// Mitsubishi GX Works2 project: Rev 1   PLC: FX3G

PROGRAM MAIN
VAR
  b0 : BOOL;  (* Start Buttom *)
  b1 : BOOL;  (* Stop Button *)
  b2 : BOOL;  (* Refference Output *)
  sm400 : BOOL;
END_VAR
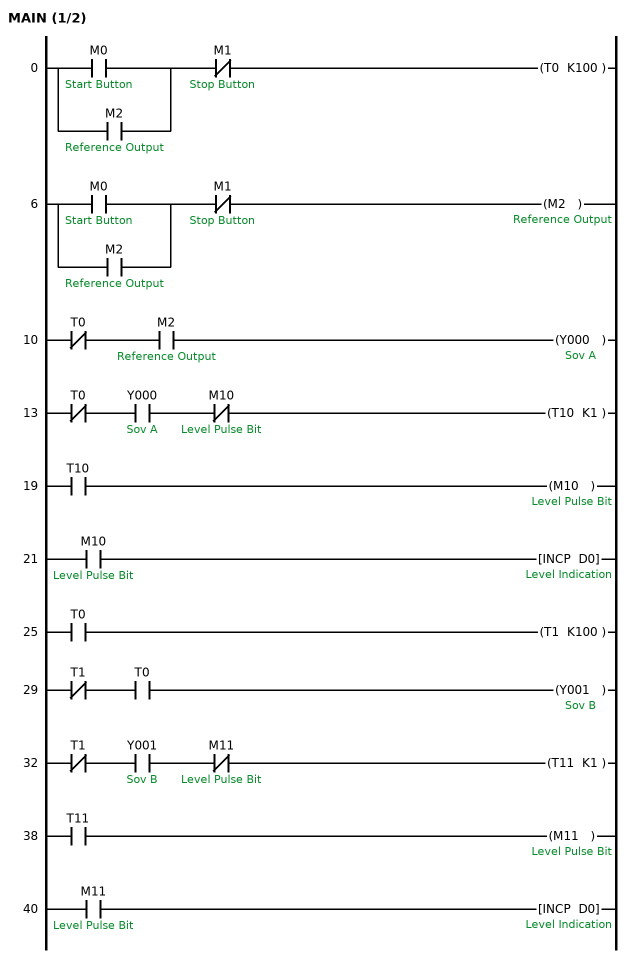
0     LD      M0  ; Start Button
      OR      M2  ; Reference Output
      ANI     M1  ; Stop Button
      OUT     T0 K100
6     LD      M0  ; Start Button
      OR      M2  ; Reference Output
      ANI     M1  ; Stop Button
      OUT     M2  ; Reference Output
10    LDI     T0
      AND     M2  ; Reference Output
      OUT     Y000  ; Sov A
13    LDI     T0
      AND     Y000  ; Sov A
      ANI     M10  ; Level Pulse Bit
      OUT     T10 K1
19    LD      T10
      OUT     M10  ; Level Pulse Bit
21    LD      M10  ; Level Pulse Bit
      INCP    D0  ; Level Indication
25    LD      T0
      OUT     T1 K100
29    LDI     T1
      AND     T0
      OUT     Y001  ; Sov B
32    LDI     T1
      AND     Y001  ; Sov B
      ANI     M11  ; Level Pulse Bit
      OUT     T11 K1
38    LD      T11
      OUT     M11  ; Level Pulse Bit
40    LD      M11  ; Level Pulse Bit
      INCP    D0
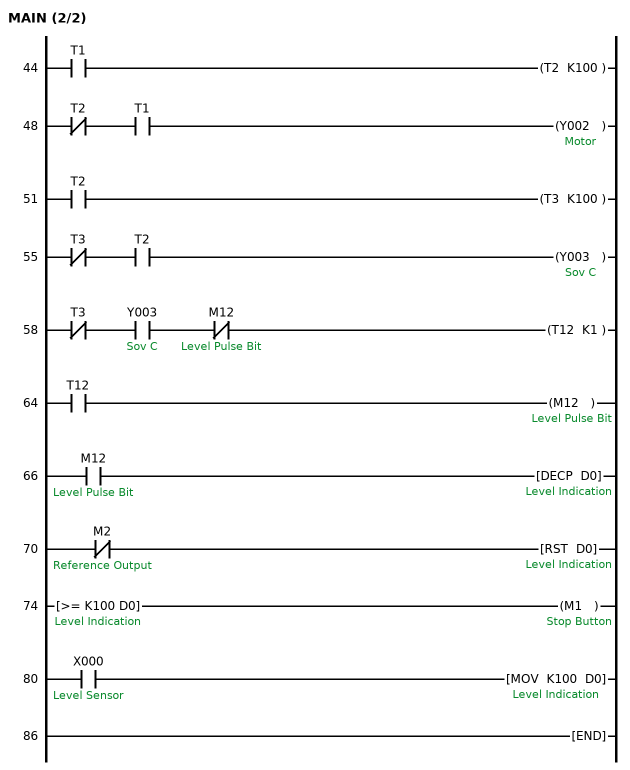
44    LD      T1
      OUT     T2 K100
48    LDI     T2
      AND     T1
      OUT     Y002  ; Motor
51    LD      T2
      OUT     T3 K100
55    LDI     T3
      AND     T2
      OUT     Y003  ; Sov C
58    LDI     T3
      AND     Y003  ; Sov C
      ANI     M12  ; Level Pulse Bit
      OUT     T12 K1
64    LD      T12
      OUT     M12  ; Level Pulse Bit
66    LD      M12  ; Level Pulse Bit
      DECP    D0
70    LDI     M2  ; Reference Output
      RST     D0  ; Level Indication
74    LD>=    K100 D0  ; Level Indication
      OUT     M1  ; Stop Button
80    LD      X000  ; Level Sensor
      MOV     K100 D0
86    END
END_PROGRAM

// device comments not shown above
Y004  ; Sov C
